FUNCTION_BLOCK T_RoboConnect_DisableNotConnected_ReturnsFalse EXTENDS T_UnitTestBase
VAR
  robot : T_MockRoboConnect;
  expected : BOOL := FALSE;
  actual : BOOL := TRUE;
END_VAR

actual := robot.Disable();
assertion.AssertEquals_BOOL(expected, actual, 'actual := robot.Disable();');
TestFinished();

END_FUNCTION_BLOCK

(* stored: Version 1.1.0.1
   POU T_TcRobot_DisableNotConnected_ReturnsFalse: Id {9337bc50-7949-4f97-b92b-8bbbe2c5dec3}, SpecialFunc None *)
